PROGRAM INTERNAL FsP_TempPlayground
VAR
END_VAR

ObjectPlayground();

METHOD PRIVATE TempPlayground
VAR_STAT
END_VAR
END_METHOD

END_PROGRAM

(* stored: Version 1.1.0.1, ProductVersion 3.1.4024.4
   POU FsP_TempPlayground: Id {796d70f3-f93a-4078-8454-4d482cd96b06}, SpecialFunc None
   Method TempPlayground: Id {381660e5-032b-42a6-9ca1-c80debbb6c20} *)
